{attribute 'linkalways'} 
{attribute 'no_explicit_call' := 'This FB is a CLASS and must be accessed using methods or properties'}
{attribute 'enable_dynamic_creation'}
FUNCTION_BLOCK _UDINT EXTENDS IntegerDatatypeBase
VAR
	localData : UDINT;
	activeData : REFERENCE TO UDINT REF= localData;
END_VAR

PROPERTY PUBLIC Address : PVOID
GET
Address := ADR(activeData);
END_GET
END_PROPERTY

METHOD PUBLIC ClearReference
VAR_INPUT
END_VAR
activeData REF= localData;
END_METHOD

METHOD PUBLIC Clone : I_Datatype
VAR
    pClone : POINTER TO _UDINT;
END_VAR
pClone := __NEW(_UDINT(InitialValue := Value));
Clone := pClone^;
END_METHOD

PROPERTY PUBLIC Datatype : T_MAXSTRING
GET
Datatype := 'UDINT';
END_GET
END_PROPERTY

METHOD FB_init : BOOL
VAR_INPUT
	bInitRetains : BOOL; // if TRUE, the retain variables are initialized (warm start / cold start)
	bInCopyCode : BOOL;  // if TRUE, the instance afterwards gets moved into the copy code (online change)
	InitialValue : UDINT;
END_VAR
localData := InitialValue;
END_METHOD

PROPERTY PUBLIC IsSigned : BOOL
GET
IsSigned := FALSE;
END_GET
END_PROPERTY

PROPERTY PUBLIC LowerBound : UDINT
GET
LowerBound := DatatypeLimits.UDINT_LOWER_LIMIT;
END_GET
END_PROPERTY

METHOD PUBLIC MakeReferenceTo
VAR_INPUT
	ReferenceTarget : REFERENCE TO UDINT;
END_VAR
activeData REF= ReferenceTarget;
END_METHOD

METHOD PROTECTED SerializeLowerbound
VAR_INPUT
	Serializer : I_Serializer;
END_VAR
Serializer.AddLint(Lowerbound);
END_METHOD

METHOD PROTECTED SerializeUpperbound
VAR_INPUT
	Serializer : I_Serializer;
END_VAR
Serializer.AddLint(Upperbound);
END_METHOD

METHOD PUBLIC SerializeWith
VAR_INPUT
	Serializer : I_Serializer;
END_VAR
Serializer.AddUdint(activeData);
END_METHOD

PROPERTY PUBLIC Size : UDINT
GET
Size := SIZEOF(activeData);
END_GET
END_PROPERTY

METHOD TryDeserializeFrom : BOOL
VAR_INPUT
	Deserializer : I_Deserializer;
	Feedback : I_DeserializerFeedback;
END_VAR
TryDeserializeFrom := Deserializer.TryGetUdint(activeData, Feedback);
END_METHOD

METHOD TryMakeReferenceTo : BOOL
VAR_INPUT
	Target : I_Datatype;
END_VAR
VAR
	pTargetData : POINTER TO UDINT;
END_VAR
IF NOT (Target.Datatype = Datatype) THEN
	RETURN;
END_IF

pTargetData := Target.Address;
activeData REF= pTargetData^;
TryMakeReferenceTo := TRUE;
END_METHOD

PROPERTY PUBLIC UpperBound : UDINT
GET
UpperBound :=  DatatypeLimits.UDINT_UPPER_LIMIT;
END_GET
END_PROPERTY

PROPERTY PUBLIC Value : UDINT
GET
Value := activeData;
END_GET
SET
activeData := Value;
END_SET
END_PROPERTY

END_FUNCTION_BLOCK

(* stored: Version 1.1.0.1, ProductVersion 3.1.4024.12
   POU _UDINT: Id {de214b7a-abf6-0651-029b-545b4ad197b9}, SpecialFunc None
   Folder Constructor: Id {f6031e1f-4c91-0c03-19d6-9dccd778de84}
   Folder Protected: Id {b4a4ec1f-eee5-0bfb-1da6-76fc7977a50b}
   Property Address: Id {68857d8d-3222-0b90-0e75-e2eb66bb20db}
   Get Get: Id {61a1346d-1ee4-0207-039a-3ea82b857df0}
   Method ClearReference: Id {d4003dc8-faec-045c-1ed5-faec3e25c908}
   Method Clone: Id {a91594eb-c5a1-00ee-1e7e-08a3745bbd8c}
   Property Datatype: Id {e58a4370-a43f-0c3b-1506-4ba8dd4cba73}
   Get Get: Id {75922675-c7d3-0967-0f21-3e86fc41d0f1}
   Method FB_init: Id {5e956179-fbc8-0ad4-0ea9-fed8c8c22844}
   Property IsSigned: Id {ec49bc0c-7554-0ac2-36ae-4d3c8ed9b112}
   Get Get: Id {206f4891-ee01-065b-133d-a0141362c602}
   Property LowerBound: Id {f53777f7-90c3-0105-1e1b-8975b43d6794}
   Get Get: Id {179ca923-a248-038c-12a8-fcb6ae6bec83}
   Method MakeReferenceTo: Id {e14dfa75-fa6e-005e-06bb-cf4d241b8273}
   Method SerializeLowerbound: Id {f7fe814c-c8bb-0bfb-3ced-aa31527809da}
   Method SerializeUpperbound: Id {a73dbac7-95d9-0a54-20e0-dc8f9493f6ac}
   Method SerializeWith: Id {fcacdb4f-c62d-011e-332d-3b0123f7a096}
   Property Size: Id {61cee6a5-3778-0cf1-1f79-086a97564373}
   Get Get: Id {076367e7-9f45-077c-2d79-b752e53ddd18}
   Method TryDeserializeFrom: Id {f19cd9a0-83c7-02a8-1341-a2192c66d5a5}
   Method TryMakeReferenceTo: Id {442e78e5-6f67-015d-386b-1d382276b680}
   Property UpperBound: Id {e93cbcbb-490f-0374-2480-a081c522d9df}
   Get Get: Id {3b776d5f-d1f4-006b-0fa9-530dd12449b5}
   Property Value: Id {93fe3d50-495a-0b74-2b8a-8f5c9ea6ca31}
   Get Get: Id {d6d0c3b9-593e-0c42-3aa5-e82b7aeb840e}
   Set Set: Id {6289f453-b93e-09bf-256e-903098ac5511} *)
